TYPE ST_NORMAL_CAM_HANDLER_HMI :
STRUCT
END_STRUCT
END_TYPE

(* stored: Version 1.1.0.1
   DUT ST_NORMAL_CAM_HANDLER_HMI: Id {093b120d-3d92-4905-b105-59148ea5566a} *)
